(* PLC project canopen_master, beremiz beremiz 1 *)
(* stored: creationDateTime 2008-06-24T18:44:00, modificationDateTime 2026-05-28T18:18:56, language en-US *)

PROGRAM test_main_slave
  VAR
    outvar AT %QW0.1.8192.0 : INT;
    invar AT %IW0.1.8193.0 : INT;
  END_VAR

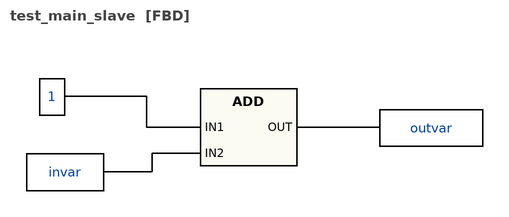
(* FBD diagram, written out as Structured Text *)
outvar := 1 + invar;
END_PROGRAM

PROGRAM test_main_master
  VAR
    PLC_OUT AT %QW0.0.2.8193.0 : INT;
    PLC_IN AT %IW0.0.2.8192.0 : INT;
  END_VAR

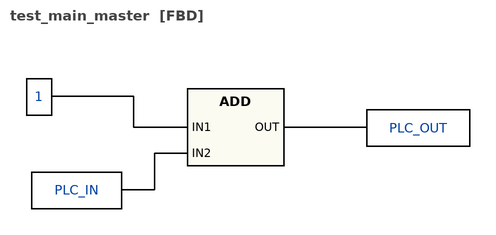
(* FBD diagram, written out as Structured Text *)
PLC_OUT := 1 + PLC_IN;
END_PROGRAM

CONFIGURATION conf
  RESOURCE res ON PLC
    TASK tache(INTERVAL := t#50ms, PRIORITY := 0);
    PROGRAM master WITH tache : test_main_master;
    PROGRAM slave WITH tache : test_main_slave;
  END_RESOURCE
END_CONFIGURATION
